// TwinCAT 3 PLC project PackMLLib
// Title: Pack ML Library
// Company: Beckhoff UK
// Author: Chris Knight
// ProjectVersion: 2.0.0.0
// ProgramVersion: 3.1.4026.15
// libraries:
//   Base Library, * (Beckhoff UK)
//   Tc2_Standard, * (Beckhoff Automation GmbH)
//   Tc3_Module, * (Beckhoff Automation GmbH)
//   Tc3_PackML_V2, * (Beckhoff Automation GmbH)
// project tree:
//   PackML/ IPmlStateMachine.TcIO, PMLStateMachine.TcPOU
//   PackML_Method_Pattern/ PML_Method_Base.TcPOU

// ---- PackML/IPmlStateMachine.TcIO
INTERFACE IPmlStateMachine

METHOD public GetCurrentMode : E_PmlProtectedUnitMode
VAR_INPUT
END_VAR
END_METHOD

METHOD GetCurrentState : E_PMLState
VAR_INPUT
END_VAR
END_METHOD

METHOD PmlModeCommand : BOOL
VAR_INPUT
	Mode : E_PMLProtectedUnitMode;
END_VAR
END_METHOD

METHOD PmlStateCommand : bool
VAR_INPUT
	Command : E_PMLCommand;
END_VAR
END_METHOD

METHOD SetStateComplete : BOOL
VAR_INPUT
END_VAR
END_METHOD

END_INTERFACE

// ---- PackML/PMLStateMachine.TcPOU
FUNCTION_BLOCK PMLStateMachine IMPLEMENTS I_Cyclic, IPmlStateMachine
VAR_INPUT
END_VAR
VAR_OUTPUT
END_VAR
VAR
	_pmlStateMachine : Tc3_PackML_V2.PML_StateMachine;
	_pmlModeMachine : Tc3_PackML_V2.PML_UnitModeManager;
	_subUnits : ARRAY[0..9] OF IPmlStateMachine;
	subUnitArray : ARRAY[0..9] OF ST_PMLSubUnitInfo;
	_SubUnitReference: ST_PMLSubUnitInfoRef;
	modeChangeTrigger : Tc2_Standard.R_TRIG;
	i: UDINT;
END_VAR

{analysis -2}

METHOD PUBLIC  Cycle : HRESULT
VAR_INPUT
END_VAR
IF _SubUnitReference.NoOfSubUnits <> 0 THEN
	FOR i := 0 TO 9 DO
		IF _subUnits[i] <> 0 THEN
			subUnitArray[i].eState := _subUnits[i].GetCurrentState();
			subUnitArray[i].Active := True;
		END_IF
	END_FOR
	_SubUnitReference.pArray := ADR(subUnitArray);
	_SubUnitReference.ArraySize := SIZEOF(subUnitArray);
END_IF

_pmlStateMachine(eMode := _pmlModeMachine.eModeStatus, stSubUnitInfoRef := _SubUnitReference);
_pmlModeMachine(eState := _pmlStateMachine.eState);
_pmlModeMachine.bExecute := FALSE;
Cycle := S_OK;
END_METHOD

METHOD PUBLIC GetCurrentMode : E_PmlProtectedUnitMode
VAR_INPUT
END_VAR
GetCurrentMode := _pmlModeMachine.eModeStatus;
END_METHOD

METHOD PUBLIC GetCurrentState : E_PMLState
VAR_INPUT
END_VAR
GetCurrentState := _pmlStateMachine.eState;
END_METHOD

METHOD PUBLIC PmlModeCommand : Bool
VAR_INPUT
	Mode : E_PMLProtectedUnitMode;
END_VAR
_pmlModeMachine.eModeCommand := Mode;
_pmlModeMachine.bExecute := TRUE;
PmlModeCommand := TRUE;
END_METHOD

METHOD PUBLIC PmlStateCommand : BOOL
VAR_INPUT
	Command : E_PMLCommand;
END_VAR
_pmlStateMachine.eCommand := Command;
PmlStateCommand := TRUE;
END_METHOD

METHOD PUBLIC RegisterSubUnit : IPmlStateMachine
VAR_INPUT
	SubUnit : IPmlStateMachine;
END_VAR
FOR i := 0 TO 9 DO
	IF _subUnits[i] = 0 THEN
		_subUnits[i] := SubUnit;
		_SubUnitReference.NoOfSubUnits := i + 1;
		EXIT;
	END_IF
END_FOR
END_METHOD

METHOD PUBLIC SetStateComplete : BOOL
VAR_INPUT
END_VAR
_pmlStateMachine.M_StateComplete();
SetStateComplete := TRUE;
END_METHOD

END_FUNCTION_BLOCK

// ---- PackML_Method_Pattern/PML_Method_Base.TcPOU
FUNCTION_BLOCK PML_Method_Base IMPLEMENTS I_Cyclic
VAR_INPUT
END_VAR
VAR_OUTPUT
END_VAR
VAR
	ipackml : IPmlStateMachine;
END_VAR

{analysis -2}

METHOD PROTECTED Aborted : BOOL
VAR_INPUT
END_VAR
Aborted := true;
END_METHOD

METHOD PROTECTED Aborting : BOOL
VAR_INPUT
END_VAR
ipackml.SetStateComplete();
Aborting := TRUE;
END_METHOD

METHOD PROTECTED Clearing : BOOL
VAR_INPUT
END_VAR
ipackml.SetStateComplete();
Clearing := TRUE;
END_METHOD

METHOD PROTECTED Completed : BOOL
VAR_INPUT
END_VAR
Completed := TRUE;
END_METHOD

METHOD PROTECTED Completing : BOOL
VAR_INPUT
END_VAR
ipackml.SetStateComplete();
Completing := TRUE;
END_METHOD

METHOD PUBLIC Cycle : HRESULT
VAR
	StateCallResult : BOOL;
END_VAR
CASE ipackml.GetCurrentState() OF
	E_PMLState.ePMLState_Clearing:
		StateCallResult := Clearing();
	E_PMLState.ePMLState_Aborted:
		StateCallResult := Aborted();
	E_PMLState.ePMLState_Aborting:
		StateCallResult := Aborting();
	E_PMLState.ePMLState_Complete:
		StateCallResult := Completed();
	E_PMLState.ePMLState_Completing:
		StateCallResult := Completing();
	E_PMLState.ePMLState_Execute:
		StateCallResult := Execute();
	E_PMLState.ePMLState_Held:
		StateCallResult := Held();
	E_PMLState.ePMLState_Holding:
		StateCallResult := Holding();
	E_PMLState.ePMLState_Idle:
		StateCallResult := Idle();
	E_PMLState.ePMLState_Resetting:
		StateCallResult := Resetting();
	E_PMLState.ePMLState_Starting:
		StateCallResult := Starting();
	E_PMLState.ePMLState_Stopped:
		StateCallResult := Stopped();
	E_PMLState.ePMLState_Stopping:
		StateCallResult := Stopping();
	E_PMLState.ePMLState_Suspended:
		StateCallResult := Suspended();
	E_PMLState.ePMLState_Suspending:
		StateCallResult := Suspending();
	E_PMLState.ePMLState_Undefined:
		StateCallResult := Undefined();
	E_PMLState.ePMLState_Unholding:
		StateCallResult := Unholding();
	E_PMLState.ePMLState_Unsuspending:
		StateCallResult := Unsuspending();
	ELSE
		Cycle := E_FAIL;
END_CASE
IF StateCallResult THEN
	Cycle := S_OK;
ELSE
	Cycle := E_FAIL;
END_IF
END_METHOD

METHOD PROTECTED Execute : BOOL
VAR_INPUT
END_VAR
Execute := true;
END_METHOD

METHOD PROTECTED Held : BOOL
VAR_INPUT
END_VAR
Held := TRUE;
END_METHOD

METHOD PROTECTED Holding : BOOL
VAR_INPUT
END_VAR
ipackml.SetStateComplete();
Holding := TRUE;
END_METHOD

METHOD PROTECTED Idle : BOOL
VAR_INPUT
END_VAR
Idle := TRUE;
END_METHOD

PROPERTY PUBLIC PackMLStateMachine : IPmlStateMachine
GET
PackMLStateMachine := ipackml;
END_GET
SET
ipackml := PackMLStateMachine;
END_SET
END_PROPERTY

METHOD PROTECTED Resetting : BOOL
VAR_INPUT
END_VAR
ipackml.SetStateComplete();
Resetting := TRUE;
END_METHOD

METHOD PROTECTED Starting : BOOL
VAR_INPUT
END_VAR
ipackml.SetStateComplete();
Starting := TRUE;
END_METHOD

METHOD PROTECTED Stopped : BOOL
VAR_INPUT
END_VAR
Stopped := TRUE;
END_METHOD

METHOD PROTECTED Stopping : BOOL
VAR_INPUT
END_VAR
ipackml.SetStateComplete();
Stopping := TRUE;
END_METHOD

METHOD PROTECTED Suspended : BOOL
VAR_INPUT
END_VAR
Suspended := TRUE;
END_METHOD

METHOD PROTECTED Suspending : BOOL
VAR_INPUT
END_VAR
ipackml.SetStateComplete();
Suspending := TRUE;
END_METHOD

METHOD PROTECTED Undefined : BOOL
VAR_INPUT
END_VAR
Undefined := TRUE;
END_METHOD

METHOD PROTECTED Unholding : BOOL
VAR_INPUT
END_VAR
ipackml.SetStateComplete();
Unholding := TRUE;
END_METHOD

METHOD PROTECTED Unsuspending : BOOL
VAR_INPUT
END_VAR
ipackml.SetStateComplete();
Unsuspending := TRUE;
END_METHOD

END_FUNCTION_BLOCK
